VAR_GLOBAL
	
	SystemON				: BOOL;
	
	LeftMotor				: AXIS_REF;
	RightMotor				: AXIS_REF;
	
	DriveTrainEnabled		: BOOL;
	
	JogLeftMotor			: BOOL;
	JogRightMotor			: BOOL;
	
	LeftLimitExceeded		: BOOL;
	RightLimitExceeded		: BOOL;
	HaltLeftMotor			: BOOL;
	HaltRightMotor			: BOOL;
	
	R100_01					: BOOL;
	R100_02					: BOOL;
	R100_03					: BOOL;
	R100_04					: BOOL;
	
END_VAR

(* stored: Version 1.1.0.1, ProductVersion 3.1.4022.7
   GVL GVL: Id {9780e9c6-3f01-408f-a62c-3bd16b7bea4b} *)
